PROGRAM MAIN
VAR
	fbArray_List_Test : FB_Array_List_Test;
	fbList_Test : FB_List_Test;
	// Add test for Array
	// Add test for Immutable list and array
	// Add test for Set
	// Add test for Immutable Set
	// Add test for Tree Map
	// Add test for Hash Map
	// Add test for Immutable Map
END_VAR

TcUnit.RUN();

END_PROGRAM

(* stored: Version 1.1.0.1, ProductVersion 3.1.4024.4
   POU MAIN: Id {17732e83-93d3-4e32-896f-74d26e2dd9ab}, SpecialFunc None *)
